{attribute 'qualified_only'} // Variable needs to be used with GVL-name
// INT: [-32768, 32767]	
// BOOL: True/False
// %Q* assigns next available memory adress in Twincat (Out)

VAR_GLOBAL
	// Digital Outputs
	bGreenLight 			AT %Q* : BOOL;	// Green light on controller
	bRedLight 				AT %Q* : BOOL;	// Red light on controller
	
	// Analog Outputs
	nValveOutput 			AT %Q* : INT;	// Valve output
	bRunning				AT %Q* : BOOL;
END_VAR

(* stored: Version 1.1.0.1
   GVL G_Output: Id {9f09a37e-4151-41e9-b303-85d293f6f5b3} *)
